// TIA Portal project "Triedenie_beden;S7-1500+TP700_Confort+OPC_UA" (V14)

(* hardware
DEVICE "S71500/ET200MP station_1"  S7-1500 station
   slot 0: "Rail_0"  Rack  6ES7 590-1***0-0AA0
   slot 1: "S7-1500"  CPU 1512C-1 PN  6ES7 512-1CK00-0AB0  V2.1
      slot 3: "CPU display_1"  6ES7591-1AA00-0AA0
DEVICE "HMI"  TP700 Comfort
   slot 0: "TP700 Comfort"  TP700 Comfort  6AV2 124-0GC01-0AX0  14.0.1.0
   slot 1: "HMI_RT_1"  TP700 Comfort  6AV2 124-0GC01-0AX0  14.0.1.0
   slot 5: "HMI.IE_CP_1"  PROFINET Interface  14.0.1.0
      slot 1: "PROFINET Interface_1"  PROFINET Interface
         slot 1: "Port_1"  Port
         slot 2: "Port_2"  Port
   slot 7: "HMI.MPI/DP_CP_1"  MPI/DP Interface  14.0.1.0
*)

// ===== PLC "S7-1500"  CPU 1512C-1 PN =====

VAR_GLOBAL   // PLC tag table "Default tag table"
   "BTN_red" AT %I13.7 : Bool;
   "BTN_green" AT %I13.6 : Bool;
   "senzor_1" AT %I13.5 : Bool;
   "senzor_2" AT %I13.4 : Bool;
   "motor_1" AT %Q7.7 : Bool;
   "motor_3_k_pasu" AT %Q7.6 : Bool;
   "motor_3_od_pasu" AT %Q7.5 : Bool;
   "motor_2_k_pasu" AT %Q7.4 : Bool;
   "motor_2_od_pasu" AT %Q7.3 : Bool;
   "solenoid_1" AT %Q7.2 : Bool;
   "solenoid_2" AT %Q7.1 : Bool;
   "LED_red" AT %Q7.0 : Bool;
   "LED_green" AT %Q6.7 : Bool;
   "stav_INIT" AT %M10.0 : Bool;
   "stav_scan" AT %M10.1 : Bool;
   "stav_mala_1" AT %M11.0 : Bool;
   "stav_mala_2" AT %M11.1 : Bool;
   "stav_mala_3" AT %M11.2 : Bool;
   "stav_mala_4" AT %M11.3 : Bool;
   "stav_mala_5" AT %M11.4 : Bool;
   "stav_mala_6" AT %M11.5 : Bool;
   "stav_mala_7" AT %M11.6 : Bool;
   "stav_mala_8" AT %M11.7 : Bool;
   "stav_velka_1" AT %M12.0 : Bool;
   "stav_velka_2" AT %M12.1 : Bool;
   "stav_velka_3" AT %M12.2 : Bool;
   "stav_velka_4" AT %M12.3 : Bool;
   "stav_velka_5" AT %M12.4 : Bool;
   "stav_velka_6" AT %M12.5 : Bool;
   "stav_velka_7" AT %M12.6 : Bool;
   "stav_velka_8" AT %M12.7 : Bool;
   "stavy_mala" AT %MB11 : Byte;
   "stavy_velka" AT %MB12 : Byte;
   "stavy" AT %MB10 : Byte;
   "stav_vyloz_male" AT %M13.0 : Bool;
   "stav_vyloz_male_1" AT %M13.1 : Bool;
   "stav_vyloz_male_2" AT %M13.2 : Bool;
   "stav_vyloz_male_trigger" AT %M13.3 : Bool;
   "stavy_vyloz_male" AT %MB13 : Byte;
   "stav_vyloz_stred" AT %M14.0 : Bool;
   "stav_vyloz_stred_1" AT %M14.1 : Bool;
   "stav_vyloz_stred_2" AT %M14.2 : Bool;
   "stav_vyloz_stredne_trigger" AT %M14.3 : Bool;
   "stavy_vyloz_stredne" AT %MB14 : Byte;
END_VAR

DATA_BLOCK "DataBlock"   // DB2
{ S7_Optimized_Access := 'TRUE' }
VERSION : 0.1
   VAR
      scan_Time_sens1 : Time;
      hold_scan_time_sens1 : Time;
      pocet_malych : Int;
      pocet_strednych : Int;
      pocet_velkych : Int;
      paleta_male_full : Bool;
      paleta_stred_full : Bool;
      paleta_male_vylozena : Bool;
      paleta_male_prec : Bool;
      paleta_stred_vylozena : Bool;
      paleta_stred_prec : Bool;
      func_paleta_male_help : Bool;
      func_paleta_stred_help : Bool;
      motor2_ON : Bool;
      motor3_ON : Bool;
      reset_citace : Bool;
      mala : Bool;
      stredna : Bool;
      velka : Bool;
   END_VAR
BEGIN
END_DATA_BLOCK

DATA_BLOCK "triedenie_DB"   // DB3
{ S7_Optimized_Access := 'TRUE' }
VERSION : 0.1
// stored: InstanceOfName triedenie
"triedenie"
BEGIN
END_DATA_BLOCK

// folder: System blocks/Program resources

DATA_BLOCK "IEC_Timer_0_DB"   // DB1
{ S7_Optimized_Access := 'TRUE' }
AUTHOR : Simatic
FAMILY : IEC
NAME : IEC_TMR
VERSION : 1.0
// stored: InstanceOfName IEC_TIMER
"IEC_TIMER"
BEGIN
END_DATA_BLOCK

DATA_BLOCK "IEC_Counter_0_DB"   // DB4
{ S7_Optimized_Access := 'TRUE' }
AUTHOR : Simatic
FAMILY : IEC
NAME : CNTR
VERSION : 1.0
// stored: InstanceOfName IEC_COUNTER
"IEC_COUNTER"
BEGIN
END_DATA_BLOCK

DATA_BLOCK "IEC_Counter_0_DB_1"   // DB5
{ S7_Optimized_Access := 'TRUE' }
AUTHOR : Simatic
FAMILY : IEC
NAME : CNTR
VERSION : 1.0
// stored: InstanceOfName IEC_COUNTER
"IEC_COUNTER"
BEGIN
END_DATA_BLOCK

DATA_BLOCK "IEC_Timer_0_DB_1"   // DB6
{ S7_Optimized_Access := 'TRUE' }
AUTHOR : Simatic
FAMILY : IEC
NAME : IEC_TMR
VERSION : 1.0
// stored: InstanceOfName IEC_TIMER
"IEC_TIMER"
BEGIN
END_DATA_BLOCK

DATA_BLOCK "IEC_Timer_0_DB_2"   // DB7
{ S7_Optimized_Access := 'TRUE' }
AUTHOR : Simatic
FAMILY : IEC
NAME : IEC_TMR
VERSION : 1.0
// stored: InstanceOfName IEC_TIMER
"IEC_TIMER"
BEGIN
END_DATA_BLOCK

DATA_BLOCK "IEC_Timer_0_DB_3"   // DB8
{ S7_Optimized_Access := 'TRUE' }
AUTHOR : Simatic
FAMILY : IEC
NAME : IEC_TMR
VERSION : 1.0
// stored: InstanceOfName IEC_TIMER
"IEC_TIMER"
BEGIN
END_DATA_BLOCK

DATA_BLOCK "IEC_Timer_0_DB_4"   // DB9
{ S7_Optimized_Access := 'TRUE' }
AUTHOR : Simatic
FAMILY : IEC
NAME : IEC_TMR
VERSION : 1.0
// stored: InstanceOfName IEC_TIMER
"IEC_TIMER"
BEGIN
END_DATA_BLOCK

DATA_BLOCK "IEC_Timer_1_DB"   // DB10
{ S7_Optimized_Access := 'TRUE' }
AUTHOR : Simatic
FAMILY : IEC
NAME : IEC_TMR
VERSION : 1.0
// stored: InstanceOfName IEC_TIMER
"IEC_TIMER"
BEGIN
END_DATA_BLOCK

DATA_BLOCK "IEC_Timer_1_DB_1"   // DB11
{ S7_Optimized_Access := 'TRUE' }
AUTHOR : Simatic
FAMILY : IEC
NAME : IEC_TMR
VERSION : 1.0
// stored: InstanceOfName IEC_TIMER
"IEC_TIMER"
BEGIN
END_DATA_BLOCK

DATA_BLOCK "IEC_Timer_1_DB_3"   // DB13
{ S7_Optimized_Access := 'TRUE' }
AUTHOR : Simatic
FAMILY : IEC
NAME : IEC_TMR
VERSION : 1.0
// stored: InstanceOfName IEC_TIMER
"IEC_TIMER"
BEGIN
END_DATA_BLOCK

DATA_BLOCK "IEC_Timer_1_DB_2"   // DB14
{ S7_Optimized_Access := 'TRUE' }
AUTHOR : Simatic
FAMILY : IEC
NAME : IEC_TMR
VERSION : 1.0
// stored: InstanceOfName IEC_TIMER
"IEC_TIMER"
BEGIN
END_DATA_BLOCK

DATA_BLOCK "IEC_Timer_2_DB"   // DB16
{ S7_Optimized_Access := 'TRUE' }
AUTHOR : Simatic
FAMILY : IEC
NAME : IEC_TMR
VERSION : 1.0
// stored: InstanceOfName IEC_TIMER
"IEC_TIMER"
BEGIN
END_DATA_BLOCK

DATA_BLOCK "IEC_Timer_2_DB_1"   // DB17
{ S7_Optimized_Access := 'TRUE' }
AUTHOR : Simatic
FAMILY : IEC
NAME : IEC_TMR
VERSION : 1.0
// stored: InstanceOfName IEC_TIMER
"IEC_TIMER"
BEGIN
END_DATA_BLOCK

DATA_BLOCK "IEC_Timer_2_DB_2"   // DB18
{ S7_Optimized_Access := 'TRUE' }
AUTHOR : Simatic
FAMILY : IEC
NAME : IEC_TMR
VERSION : 1.0
// stored: InstanceOfName IEC_TIMER
"IEC_TIMER"
BEGIN
END_DATA_BLOCK

DATA_BLOCK "IEC_Timer_2_DB_3"   // DB19
{ S7_Optimized_Access := 'TRUE' }
AUTHOR : Simatic
FAMILY : IEC
NAME : IEC_TMR
VERSION : 1.0
// stored: InstanceOfName IEC_TIMER
"IEC_TIMER"
BEGIN
END_DATA_BLOCK

// folder: (top level)

FUNCTION_BLOCK "triedenie"   // FB1, LAD
{ S7_Optimized_Access := 'TRUE' }
VERSION : 0.1
// V tomto bloku prebieha
   VAR_TEMP   // added for the SCL form of the ladder/FBD networks
      _w1 : Bool;
   END_VAR
BEGIN

REGION Network 1: Ak sú všetky stavy v 0 setni stav INIT
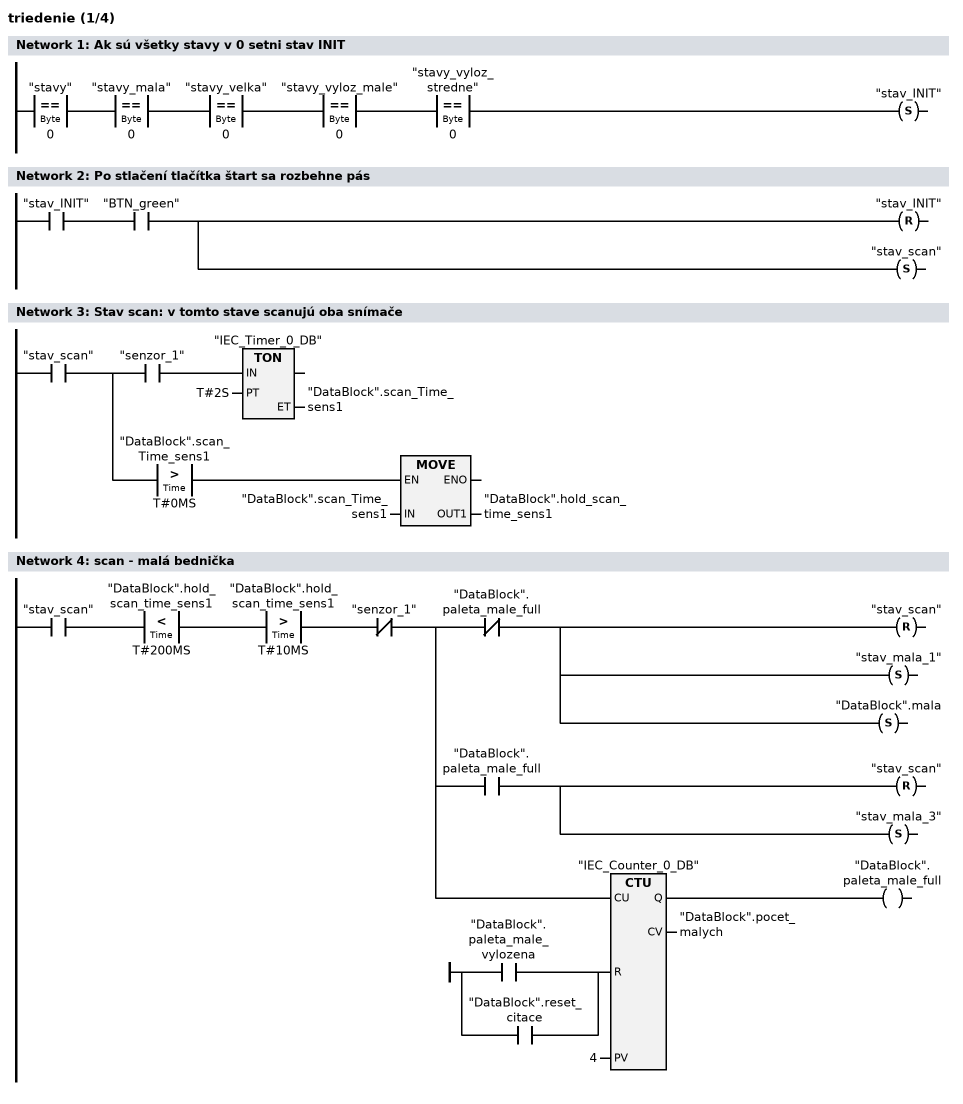
   RUNG wire#powerrail
      { S7_Templates := "SrcType := Byte" } EQ_Contact(in1 := "stavy", in2 := 0)
      { S7_Templates := "SrcType := Byte" } EQ_Contact(in1 := "stavy_mala", in2 := 0)
      { S7_Templates := "SrcType := Byte" } EQ_Contact(in1 := "stavy_velka", in2 := 0)
      { S7_Templates := "SrcType := Byte" } EQ_Contact(in1 := "stavy_vyloz_male", in2 := 0)
      { S7_Templates := "SrcType := Byte" } EQ_Contact(in1 := "stavy_vyloz_stredne", in2 := 0)
      S_Coil( "stav_INIT" )
   END_RUNG
   // the same network as SCL:
   IF ("stavy" = 0) AND ("stavy_mala" = 0) AND ("stavy_velka" = 0) AND ("stavy_vyloz_male" = 0) AND ("stavy_vyloz_stredne" = 0) THEN
       "stav_INIT" := TRUE;
   END_IF;
END_REGION

REGION Network 2: Po stlačení tlačítka štart sa rozbehne pás
   RUNG wire#powerrail
      Contact( "stav_INIT" )
      Contact( "BTN_green" )
      wire#w1
      R_Coil( "stav_INIT" )
   END_RUNG
   RUNG wire#w1
      S_Coil( "stav_scan" )
   END_RUNG
   // the same network as SCL:
   #_w1 := "stav_INIT" AND "BTN_green";
   IF #_w1 THEN
       "stav_INIT" := FALSE;
       "stav_scan" := TRUE;
   END_IF;
END_REGION

REGION Network 3: Stav scan: v tomto stave scanujú oba snímače
   "IEC_Timer_0_DB".TON(IN := "stav_scan" AND "senzor_1", PT := T#2S, ET => "DataBlock".scan_Time_sens1);
   IF "stav_scan" AND ("DataBlock".scan_Time_sens1 > T#0MS) THEN
       "DataBlock".hold_scan_time_sens1 := "DataBlock".scan_Time_sens1;
   END_IF;
END_REGION

REGION Network 4: scan - malá bednička
   #_w1 := "stav_scan" AND ("DataBlock".hold_scan_time_sens1 < T#200MS) AND ("DataBlock".hold_scan_time_sens1 > T#10MS) AND NOT "senzor_1";
   IF #_w1 AND NOT "DataBlock".paleta_male_full THEN
       "stav_scan" := FALSE;
       "stav_mala_1" := TRUE;
       "DataBlock".mala := TRUE;
   END_IF;
   IF #_w1 AND "DataBlock".paleta_male_full THEN
       "stav_scan" := FALSE;
       "stav_mala_3" := TRUE;
   END_IF;
   "IEC_Counter_0_DB".CTU(CU := #_w1,
                          R := "DataBlock".paleta_male_vylozena OR "DataBlock".reset_citace,
                          PV := 4,
                          CV => "DataBlock".pocet_malych);
   "DataBlock".paleta_male_full := "IEC_Counter_0_DB".Q;
END_REGION

REGION Network 5: scan - stredná bednička
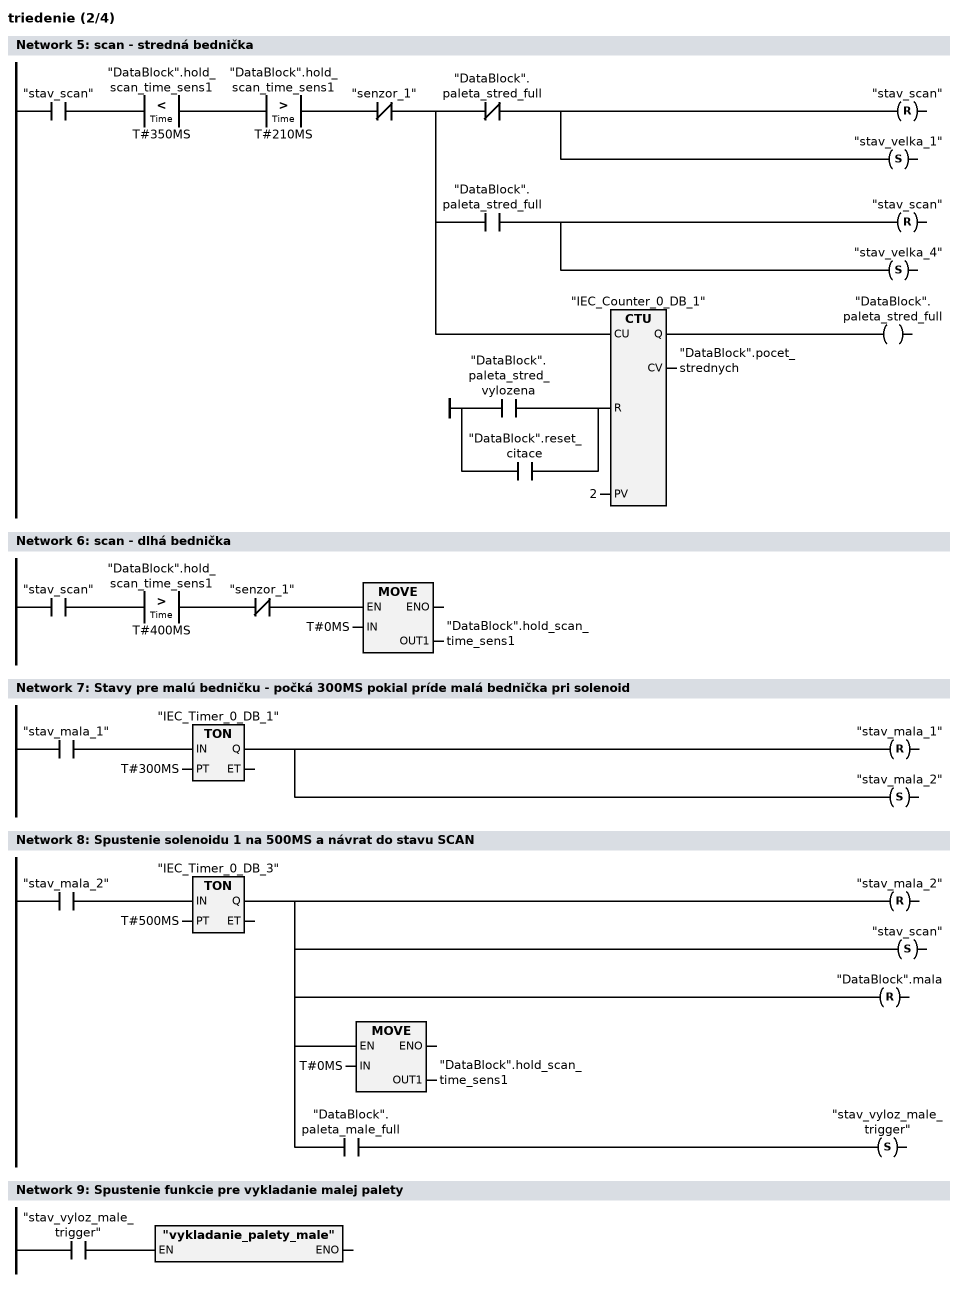
   #_w1 := "stav_scan" AND ("DataBlock".hold_scan_time_sens1 < T#350MS) AND ("DataBlock".hold_scan_time_sens1 > T#210MS) AND NOT "senzor_1";
   IF #_w1 AND NOT "DataBlock".paleta_stred_full THEN
       "stav_scan" := FALSE;
       "stav_velka_1" := TRUE;
   END_IF;
   IF #_w1 AND "DataBlock".paleta_stred_full THEN
       "stav_scan" := FALSE;
       "stav_velka_4" := TRUE;
   END_IF;
   "IEC_Counter_0_DB_1".CTU(CU := #_w1,
                           R := "DataBlock".paleta_stred_vylozena OR "DataBlock".reset_citace,
                           PV := 2,
                           CV => "DataBlock".pocet_strednych);
   "DataBlock".paleta_stred_full := "IEC_Counter_0_DB_1".Q;
END_REGION

REGION Network 6: scan - dlhá bednička
   RUNG wire#powerrail
      Contact( "stav_scan" )
      { S7_Templates := "SrcType := Time" } GT_Contact(in1 := "DataBlock".hold_scan_time_sens1, in2 := T#400MS)
      I_Contact( "senzor_1" )
      Move(in := T#0MS, out1 => "DataBlock".hold_scan_time_sens1)
   END_RUNG
   // the same network as SCL:
   IF "stav_scan" AND ("DataBlock".hold_scan_time_sens1 > T#400MS) AND NOT "senzor_1" THEN
       "DataBlock".hold_scan_time_sens1 := T#0MS;
   END_IF;
END_REGION

REGION Network 7: Stavy pre malú bedničku - počká 300MS pokial príde malá bednička pri solenoid
   "IEC_Timer_0_DB_1".TON(IN := "stav_mala_1", PT := T#300MS);
   IF "IEC_Timer_0_DB_1".Q THEN
       "stav_mala_1" := FALSE;
       "stav_mala_2" := TRUE;
   END_IF;
END_REGION

REGION Network 8: Spustenie solenoidu 1 na 500MS a návrat do stavu SCAN
   "IEC_Timer_0_DB_3".TON(IN := "stav_mala_2", PT := T#500MS);
   IF "IEC_Timer_0_DB_3".Q THEN
       "stav_mala_2" := FALSE;
       "stav_scan" := TRUE;
       "DataBlock".mala := FALSE;
       "DataBlock".hold_scan_time_sens1 := T#0MS;
   END_IF;
   IF "IEC_Timer_0_DB_3".Q AND "DataBlock".paleta_male_full THEN "stav_vyloz_male_trigger" := TRUE; END_IF;
END_REGION

REGION Network 9: Spustenie funkcie pre vykladanie malej palety
   RUNG wire#powerrail
      Contact( "stav_vyloz_male_trigger" )
      "vykladanie_palety_male"()
   END_RUNG
   // the same network as SCL:
   IF "stav_vyloz_male_trigger" THEN "vykladanie_palety_male"(); END_IF;
END_REGION

REGION Network 10: V tomto stave čakám na malú paletu
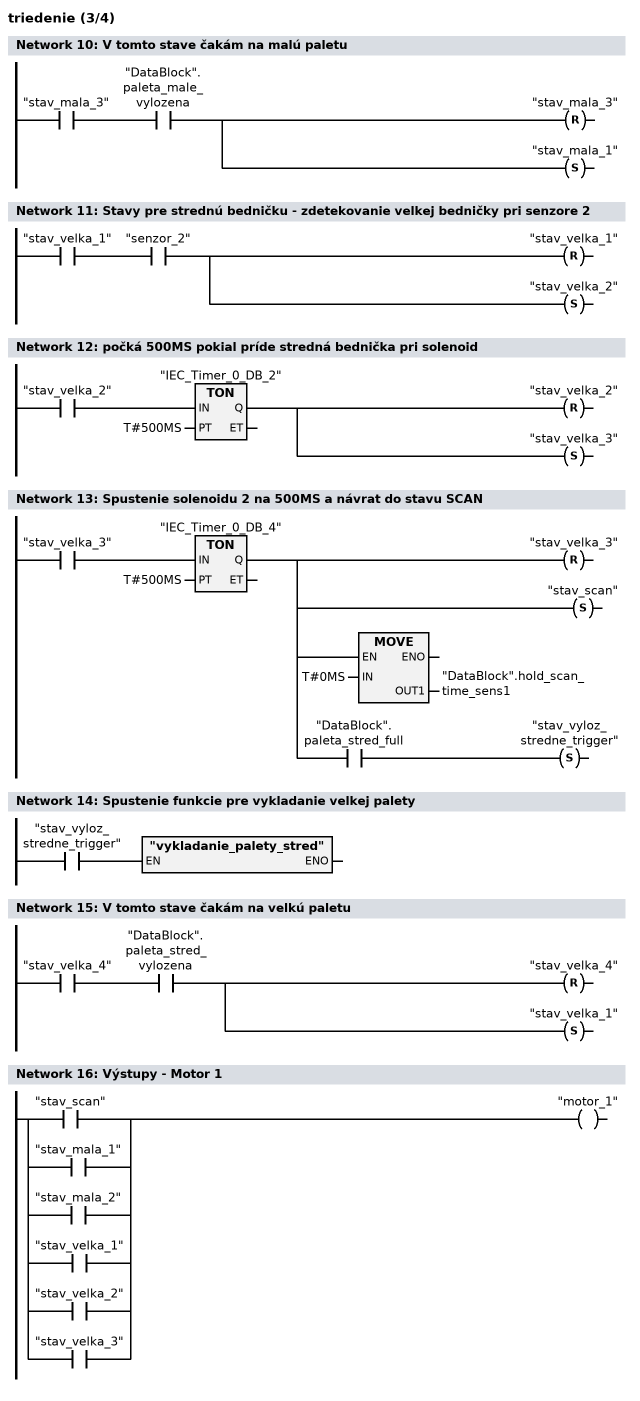
   RUNG wire#powerrail
      Contact( "stav_mala_3" )
      Contact( "DataBlock".paleta_male_vylozena )
      wire#w1
      R_Coil( "stav_mala_3" )
   END_RUNG
   RUNG wire#w1
      S_Coil( "stav_mala_1" )
   END_RUNG
   // the same network as SCL:
   #_w1 := "stav_mala_3" AND "DataBlock".paleta_male_vylozena;
   IF #_w1 THEN
       "stav_mala_3" := FALSE;
       "stav_mala_1" := TRUE;
   END_IF;
END_REGION

REGION Network 11: Stavy pre strednú bedničku - zdetekovanie velkej bedničky pri senzore 2
   RUNG wire#powerrail
      Contact( "stav_velka_1" )
      Contact( "senzor_2" )
      wire#w1
      R_Coil( "stav_velka_1" )
   END_RUNG
   RUNG wire#w1
      S_Coil( "stav_velka_2" )
   END_RUNG
   // the same network as SCL:
   #_w1 := "stav_velka_1" AND "senzor_2";
   IF #_w1 THEN
       "stav_velka_1" := FALSE;
       "stav_velka_2" := TRUE;
   END_IF;
END_REGION

REGION Network 12: počká 500MS pokial príde stredná bednička pri solenoid
   "IEC_Timer_0_DB_2".TON(IN := "stav_velka_2", PT := T#500MS);
   IF "IEC_Timer_0_DB_2".Q THEN
       "stav_velka_2" := FALSE;
       "stav_velka_3" := TRUE;
   END_IF;
END_REGION

REGION Network 13: Spustenie solenoidu 2 na 500MS a návrat do stavu SCAN
   "IEC_Timer_0_DB_4".TON(IN := "stav_velka_3", PT := T#500MS);
   IF "IEC_Timer_0_DB_4".Q THEN
       "stav_velka_3" := FALSE;
       "stav_scan" := TRUE;
       "DataBlock".hold_scan_time_sens1 := T#0MS;
   END_IF;
   IF "IEC_Timer_0_DB_4".Q AND "DataBlock".paleta_stred_full THEN
       "stav_vyloz_stredne_trigger" := TRUE;
   END_IF;
END_REGION

REGION Network 14: Spustenie funkcie pre vykladanie velkej palety
   RUNG wire#powerrail
      Contact( "stav_vyloz_stredne_trigger" )
      "vykladanie_palety_stred"()
   END_RUNG
   // the same network as SCL:
   IF "stav_vyloz_stredne_trigger" THEN "vykladanie_palety_stred"(); END_IF;
END_REGION

REGION Network 15: V tomto stave čakám na velkú paletu
   RUNG wire#powerrail
      Contact( "stav_velka_4" )
      Contact( "DataBlock".paleta_stred_vylozena )
      wire#w1
      R_Coil( "stav_velka_4" )
   END_RUNG
   RUNG wire#w1
      S_Coil( "stav_velka_1" )
   END_RUNG
   // the same network as SCL:
   #_w1 := "stav_velka_4" AND "DataBlock".paleta_stred_vylozena;
   IF #_w1 THEN
       "stav_velka_4" := FALSE;
       "stav_velka_1" := TRUE;
   END_IF;
END_REGION

REGION Network 16: Výstupy - Motor 1
   RUNG wire#powerrail
      Contact( "stav_scan" )
      wire#w1
      Coil( "motor_1" )
   END_RUNG
   RUNG wire#powerrail
      Contact( "stav_mala_1" )
   END_RUNG wire#w1
   RUNG wire#powerrail
      Contact( "stav_mala_2" )
   END_RUNG wire#w1
   RUNG wire#powerrail
      Contact( "stav_velka_1" )
   END_RUNG wire#w1
   RUNG wire#powerrail
      Contact( "stav_velka_2" )
   END_RUNG wire#w1
   RUNG wire#powerrail
      Contact( "stav_velka_3" )
   END_RUNG wire#w1
   // the same network as SCL:
   "motor_1" := "stav_scan" OR "stav_mala_1" OR "stav_mala_2" OR "stav_velka_1" OR "stav_velka_2" OR "stav_velka_3";
END_REGION

REGION Network 17: Výstupy - Solenoid 1
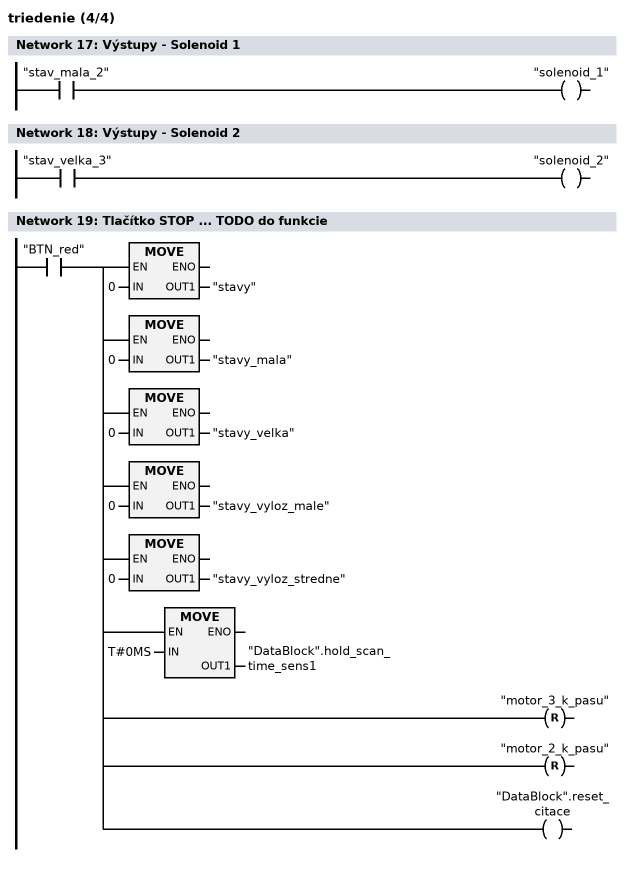
   RUNG wire#powerrail
      Contact( "stav_mala_2" )
      Coil( "solenoid_1" )
   END_RUNG
   // the same network as SCL:
   "solenoid_1" := "stav_mala_2";
END_REGION

REGION Network 18: Výstupy - Solenoid 2
   RUNG wire#powerrail
      Contact( "stav_velka_3" )
      Coil( "solenoid_2" )
   END_RUNG
   // the same network as SCL:
   "solenoid_2" := "stav_velka_3";
END_REGION

REGION Network 19: Tlačítko STOP ... TODO do funkcie
   RUNG wire#powerrail
      Contact( "BTN_red" )
      wire#w1
      Move(in := 0, out1 => "stavy")
   END_RUNG
   RUNG wire#w1
      Move(in := 0, out1 => "stavy_mala")
   END_RUNG
   RUNG wire#w1
      Move(in := 0, out1 => "stavy_velka")
   END_RUNG
   RUNG wire#w1
      Move(in := 0, out1 => "stavy_vyloz_male")
   END_RUNG
   RUNG wire#w1
      Move(in := 0, out1 => "stavy_vyloz_stredne")
   END_RUNG
   RUNG wire#w1
      Move(in := T#0MS, out1 => "DataBlock".hold_scan_time_sens1)
   END_RUNG
   RUNG wire#w1
      R_Coil( "motor_3_k_pasu" )
   END_RUNG
   RUNG wire#w1
      R_Coil( "motor_2_k_pasu" )
   END_RUNG
   RUNG wire#w1
      Coil( "DataBlock".reset_citace )
   END_RUNG
   // the same network as SCL:
   IF "BTN_red" THEN
       "stavy" := 0;
       "stavy_mala" := 0;
       "stavy_velka" := 0;
       "stavy_vyloz_male" := 0;
       "stavy_vyloz_stredne" := 0;
       "DataBlock".hold_scan_time_sens1 := T#0MS;
       "motor_3_k_pasu" := FALSE;
       "motor_2_k_pasu" := FALSE;
   END_IF;
   "DataBlock".reset_citace := "BTN_red";
END_REGION
END_FUNCTION_BLOCK

FUNCTION "vykladanie_palety_male" : Void   // FC1, LAD
{ S7_Optimized_Access := 'TRUE' }
VERSION : 0.1
   VAR_TEMP   // added for the SCL form of the ladder/FBD networks
      _w1 : Bool;
   END_VAR
BEGIN

REGION Network 1: funkcia sa spustí na nábežnú hranu
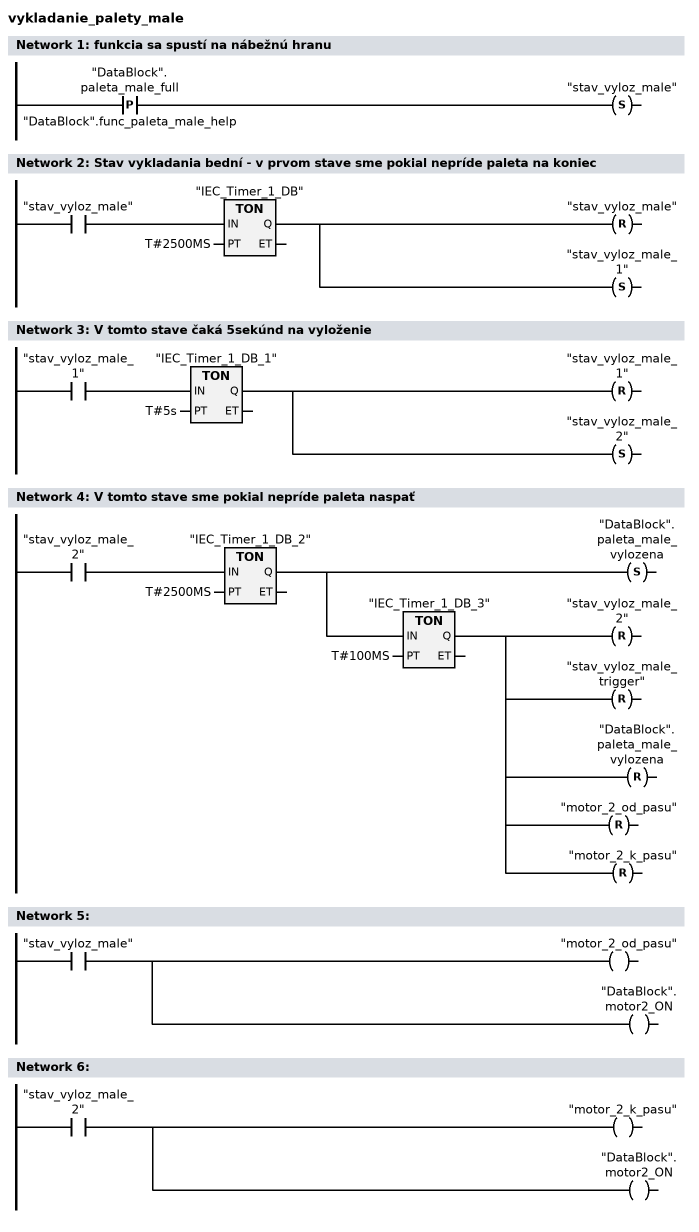
   RUNG wire#powerrail
      P_Contact(operand := "DataBlock".paleta_male_full, bit := "DataBlock".func_paleta_male_help)
      S_Coil( "stav_vyloz_male" )
   END_RUNG
   // the same network as SCL:
   #_w1 := "DataBlock".paleta_male_full AND NOT "DataBlock".func_paleta_male_help;   // rising edge of "DataBlock".paleta_male_full
   "DataBlock".func_paleta_male_help := "DataBlock".paleta_male_full;
   IF #_w1 THEN "stav_vyloz_male" := TRUE; END_IF;
END_REGION

REGION Network 2: Stav vykladania bední - v prvom stave sme pokial nepríde paleta na koniec
   "IEC_Timer_1_DB".TON(IN := "stav_vyloz_male", PT := T#2500MS);
   IF "IEC_Timer_1_DB".Q THEN
       "stav_vyloz_male" := FALSE;
       "stav_vyloz_male_1" := TRUE;
   END_IF;
END_REGION

REGION Network 3: V tomto stave čaká 5sekúnd na vyloženie
   "IEC_Timer_1_DB_1".TON(IN := "stav_vyloz_male_1", PT := T#5s);
   IF "IEC_Timer_1_DB_1".Q THEN
       "stav_vyloz_male_1" := FALSE;
       "stav_vyloz_male_2" := TRUE;
   END_IF;
END_REGION

REGION Network 4: V tomto stave sme pokial nepríde paleta naspať
   "IEC_Timer_1_DB_2".TON(IN := "stav_vyloz_male_2", PT := T#2500MS);
   IF "IEC_Timer_1_DB_2".Q THEN "DataBlock".paleta_male_vylozena := TRUE; END_IF;
   "IEC_Timer_1_DB_3".TON(IN := "IEC_Timer_1_DB_2".Q, PT := T#100MS);
   IF "IEC_Timer_1_DB_3".Q THEN
       "stav_vyloz_male_2" := FALSE;
       "stav_vyloz_male_trigger" := FALSE;
       "DataBlock".paleta_male_vylozena := FALSE;
       "motor_2_od_pasu" := FALSE;
       "motor_2_k_pasu" := FALSE;
   END_IF;
END_REGION

REGION Network 5
   RUNG wire#powerrail
      Contact( "stav_vyloz_male" )
      wire#w1
      Coil( "motor_2_od_pasu" )
   END_RUNG
   RUNG wire#w1
      Coil( "DataBlock".motor2_ON )
   END_RUNG
   // the same network as SCL:
   "motor_2_od_pasu" := "stav_vyloz_male";
   "DataBlock".motor2_ON := "stav_vyloz_male";
END_REGION

REGION Network 6
   RUNG wire#powerrail
      Contact( "stav_vyloz_male_2" )
      wire#w1
      Coil( "motor_2_k_pasu" )
   END_RUNG
   RUNG wire#w1
      Coil( "DataBlock".motor2_ON )
   END_RUNG
   // the same network as SCL:
   "motor_2_k_pasu" := "stav_vyloz_male_2";
   "DataBlock".motor2_ON := "stav_vyloz_male_2";
END_REGION
END_FUNCTION

FUNCTION "vykladanie_palety_stred" : Void   // FC2, LAD
{ S7_Optimized_Access := 'TRUE' }
VERSION : 0.1
   VAR_TEMP   // added for the SCL form of the ladder/FBD networks
      _w1 : Bool;
   END_VAR
BEGIN

REGION Network 1
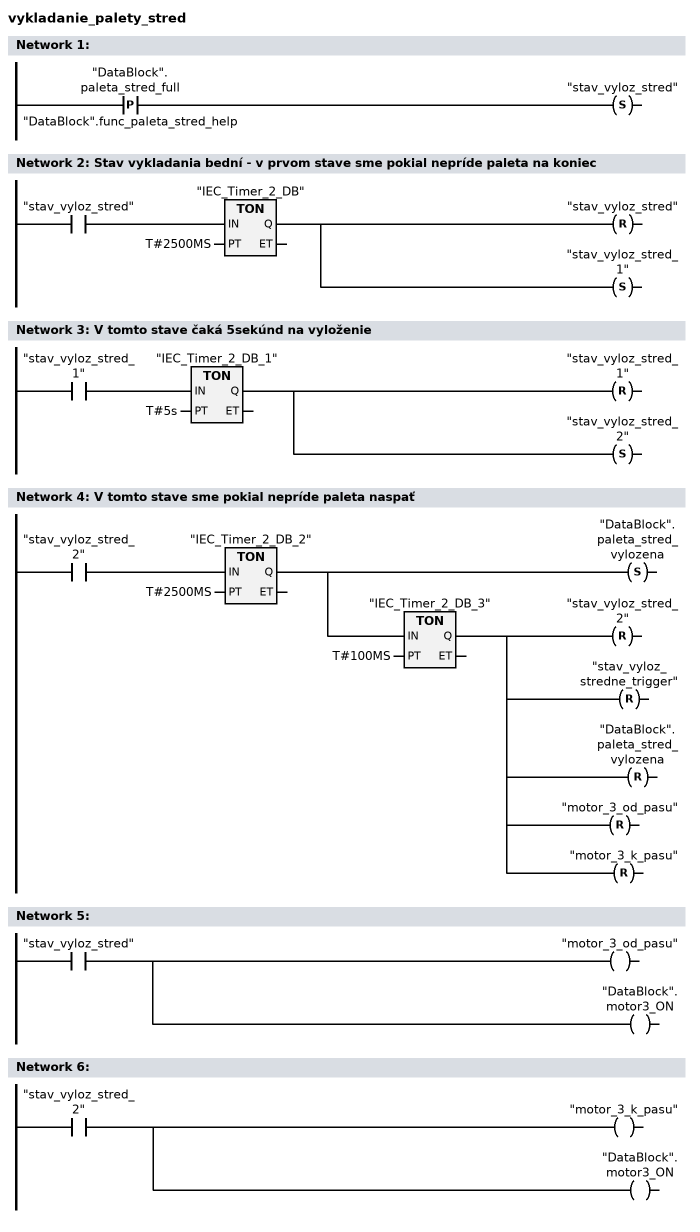
   RUNG wire#powerrail
      P_Contact(operand := "DataBlock".paleta_stred_full, bit := "DataBlock".func_paleta_stred_help)
      S_Coil( "stav_vyloz_stred" )
   END_RUNG
   // the same network as SCL:
   #_w1 := "DataBlock".paleta_stred_full AND NOT "DataBlock".func_paleta_stred_help;   // rising edge of "DataBlock".paleta_stred_full
   "DataBlock".func_paleta_stred_help := "DataBlock".paleta_stred_full;
   IF #_w1 THEN "stav_vyloz_stred" := TRUE; END_IF;
END_REGION

REGION Network 2: Stav vykladania bední - v prvom stave sme pokial nepríde paleta na koniec
   "IEC_Timer_2_DB".TON(IN := "stav_vyloz_stred", PT := T#2500MS);
   IF "IEC_Timer_2_DB".Q THEN
       "stav_vyloz_stred" := FALSE;
       "stav_vyloz_stred_1" := TRUE;
   END_IF;
END_REGION

REGION Network 3: V tomto stave čaká 5sekúnd na vyloženie
   "IEC_Timer_2_DB_1".TON(IN := "stav_vyloz_stred_1", PT := T#5s);
   IF "IEC_Timer_2_DB_1".Q THEN
       "stav_vyloz_stred_1" := FALSE;
       "stav_vyloz_stred_2" := TRUE;
   END_IF;
END_REGION

REGION Network 4: V tomto stave sme pokial nepríde paleta naspať
   "IEC_Timer_2_DB_2".TON(IN := "stav_vyloz_stred_2", PT := T#2500MS);
   IF "IEC_Timer_2_DB_2".Q THEN "DataBlock".paleta_stred_vylozena := TRUE; END_IF;
   "IEC_Timer_2_DB_3".TON(IN := "IEC_Timer_2_DB_2".Q, PT := T#100MS);
   IF "IEC_Timer_2_DB_3".Q THEN
       "stav_vyloz_stred_2" := FALSE;
       "stav_vyloz_stredne_trigger" := FALSE;
       "DataBlock".paleta_stred_vylozena := FALSE;
       "motor_3_od_pasu" := FALSE;
       "motor_3_k_pasu" := FALSE;
   END_IF;
END_REGION

REGION Network 5
   RUNG wire#powerrail
      Contact( "stav_vyloz_stred" )
      wire#w1
      Coil( "motor_3_od_pasu" )
   END_RUNG
   RUNG wire#w1
      Coil( "DataBlock".motor3_ON )
   END_RUNG
   // the same network as SCL:
   "motor_3_od_pasu" := "stav_vyloz_stred";
   "DataBlock".motor3_ON := "stav_vyloz_stred";
END_REGION

REGION Network 6
   RUNG wire#powerrail
      Contact( "stav_vyloz_stred_2" )
      wire#w1
      Coil( "motor_3_k_pasu" )
   END_RUNG
   RUNG wire#w1
      Coil( "DataBlock".motor3_ON )
   END_RUNG
   // the same network as SCL:
   "motor_3_k_pasu" := "stav_vyloz_stred_2";
   "DataBlock".motor3_ON := "stav_vyloz_stred_2";
END_REGION
END_FUNCTION

ORGANIZATION_BLOCK "Main"   // OB1, LAD, ProgramCycle
TITLE = "Main Program Sweep (Cycle)"
{ S7_Optimized_Access := 'TRUE' }
VERSION : 0.1
   VAR_INPUT
      Initial_Call : Bool;   // Initial call of this OB
      Remanence : Bool;   // =True, if remanent data are available
   END_VAR
BEGIN

REGION Network 1
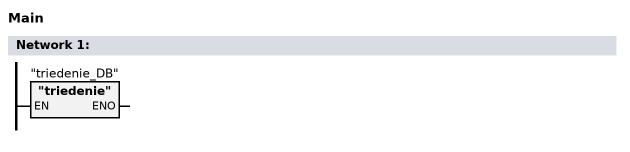
   RUNG wire#powerrail
      "triedenie_DB"()
   END_RUNG
   // the same network as SCL:
   "triedenie_DB"();   // "triedenie"
END_REGION
END_ORGANIZATION_BLOCK

(* ===== HMI "HMI_RT_1" =====
system functions are stored by id; their names below are inferred from use
connection "HMI_Connection_1": ETHERNET, S7_1500_OMS

HMI tags "Data"
   "pocet_malych" : Int = PLC DataBlock.pocet_malych AT %DB1.DBW0, 1 s
   "pocet_strednych" : Int = PLC DataBlock.pocet_strednych AT %DB1.DBW0, 1 s
   "pocet_velkych" : Int = PLC DataBlock.pocet_velkych AT %DB1.DBW0, 1 s
   "mala" : Bool = PLC DataBlock.mala AT %DB1.DBX0.0, 1 s

HMI tags "Outputs-Inputs"
   "motor_1" : Bool = PLC motor_1 AT %Q7.7, 1 s
   "motor_2_k_pasu" : Bool = PLC motor_2_k_pasu AT %Q7.4, 1 s
   "motor_2_od_pasu" : Bool = PLC motor_2_od_pasu AT %Q7.3, 1 s
   "motor_3_k_pasu" : Bool = PLC motor_3_od_pasu AT %Q7.5, 1 s
   "motor_3_od_pasu" : Bool = PLC motor_3_od_pasu AT %Q7.5, 1 s
   "motor2_on" : Bool = PLC DataBlock.motor2_ON AT %DB1.DBX0.0, 1 s
   "motor3_on" : Bool = PLC DataBlock.motor3_ON AT %DB1.DBX0.0, 1 s
   "sensor2" : Bool = PLC senzor_2 AT %I13.4, 1 s
   "sensor1" : Bool = PLC senzor_1 AT %I13.5, 1 s
   "solenoid1" : Bool = PLC solenoid_1 AT %Q7.2, 1 s
   "solenoid2" : Bool = PLC solenoid_2 AT %Q7.1, 1 s
   "btn_stop" : Bool = PLC BTN_red AT %I13.7, 1 s
   "btn_start" : Bool = PLC BTN_green AT %I13.6, 1 s

screen "Main_screen" 800x480
   GraphicView "conveyor_2" at 361,213 size 100x250; Picture "conveyor_2"
   GraphicView "conveyor_3" at 128,213 size 100x250; Picture "conveyor_2"
   GraphicView "conveyor_1" at -10,150 size 694x80; Picture "conveyor_1"
   GraphicView "motor_3" at 51,397 size 111x59; Picture "motor_3"
   Circle "Circle_motor3_ON" at 75,414 size 24x24
      Appearance <- "motor3_on"
   GraphicView "motor_2" at 285,397 size 111x59; Picture "motor_3"
   Circle "Circle_motor2_ON" at 309,415 size 24x24
      Appearance <- "motor2_on"
   GraphicView "Solenoid1_ON" at 381,16 size 73x168; Picture "solenoid stredny"
      Visibility <- "solenoid1"
   GraphicView "Solenoid1_OFF" at 382,16 size 73x154; Picture "solenoid kratky"
      Visibility <- "solenoid1"
   GraphicView "Sensor1_ON" at 485,91 size 115x152; Picture "snimacLong"
      Visibility <- "sensor1"
   GraphicView "Sensor1_OFF" at 485,92 size 115x97; Picture "snimacShort"
      Visibility <- "sensor1"
   GraphicView "Sensor2_OFF" at 232,90 size 115x97; Picture "snimacShort"
      Visibility <- "sensor2"
   GraphicView "Sensor2_ON" at 232,89 size 115x152; Picture "snimacLong"
      Visibility <- "sensor2"
   GraphicView "Solenoid2_ON" at 150,16 size 73x168; Picture "solenoid stredny"
      Visibility <- "solenoid2"
   GraphicView "Solenoid2_OFF" at 150,16 size 73x154; Picture "solenoid kratky"
      Visibility <- "solenoid2"
   GraphicView "Graphic view_1" at 382,264 size 32x36; Picture "g9445"
   GraphicView "Graphic view_3" at 414,264 size 32x36; Picture "g9445"
   GraphicView "Graphic view_4" at 142,227 size 72x77; Picture "paleta"
   GraphicView "Graphic view_6" at 376,227 size 72x77; Picture "paleta"
   Group "solenoid 2" at 150,16 size 73x168; Picture "solenoid stredny"
   Group "solenoid 1" at 381,16 size 74x168; Picture "solenoid stredny"
   Button "btn_start" at 632,304 size 163x49; TextOff 'START'
      on Press: InvertBit("btn_start")
      on Release: InvertBit("btn_start")
   Button "btn_stop" at 632,360 size 163x49; TextOff 'STOP'
      on Press: InvertBit("btn_stop")
      on Release: InvertBit("btn_stop")
   IOField "pocet_malych" at 328,232 size 33x32; FormatPattern 99
      ProcessValue <- "pocet_malych"
   IOField "pocet_strednych" at 96,232 size 33x32; FormatPattern 99
      ProcessValue <- "pocet_strednych"
   Button "btn_statistics" at 630,420 size 160x50; TextOff 'STATISTYKY'
      on Click: ActivateScreen("statistics", 0)
   Group "sensor 1" at 485,91 size 115x152; Picture "snimacLong"
   Group "sensor 2" at 232,89 size 115x152; Picture "snimacShort"
   GraphicView "motor_1" at 605,89 size 62x90; Picture "motor"
   Group "motor 3" at 51,397 size 111x59; Picture "motor_3"
   Group "motor 2" at 285,397 size 111x59; Picture "motor_3"
   Group "conveyors" at -10,150 size 694x313; Picture "conveyor_2"

screen "statistics" 800x480
   Button "Button_1" at 610,410 size 180x60; TextOff 'MAIN SCREEN'
      on Click: ActivateScreen("Main_screen", 0)
*)